PROGRAM PRG_GMD
VAR
END_VAR


// PIP_Gamma Pumps

fb_PCPM3B_PIP_1(i_stGauge := fb_IM2K0_XTES_GCC_1.PG);

// FB_MKS317

fb_EM1K0_GMD_GPI_10(PG=>);
fb_EM1K0_GMD_GPI_40(PG=>);
fb_EM1K0_GMD_GPI_70(PG=>);
fb_IM2K0_XTES_GPI_1(PG=>);
fb_TV1K0_GAS_GPI_1(PG=>);

// FB_PTM_TwisTorr

fb_EM1K0_GMD_PTM_10(i_xExtILKOk := TRUE);
fb_EM1K0_GMD_PTM_20(i_xExtILKOk := TRUE);
fb_EM1K0_GMD_PTM_30(i_xExtILKOk := TRUE);
fb_EM1K0_GMD_PTM_40(i_xExtILKOk := TRUE);
fb_EM1K0_GMD_PTM_50(i_xExtILKOk := TRUE);
fb_EM1K0_GMD_PTM_60(i_xExtILKOk := TRUE);
fb_EM1K0_GMD_PTM_70(i_xExtILKOk := TRUE);

// FB_VRC

fb_EM1K0_GMD_VRC_10(i_xExtILK_OK := TRUE, i_xOverrideMode := xSystemOverrideMode);
fb_EM1K0_GMD_VRC_20(i_xExtILK_OK := TRUE, i_xOverrideMode := xSystemOverrideMode);
fb_EM1K0_GMD_VRC_30(i_xExtILK_OK := TRUE, i_xOverrideMode := xSystemOverrideMode);
fb_EM1K0_GMD_VRC_50(i_xExtILK_OK := TRUE, i_xOverrideMode := xSystemOverrideMode);
fb_EM1K0_GMD_VRC_60(i_xExtILK_OK := TRUE, i_xOverrideMode := xSystemOverrideMode);
fb_EM1K0_GMD_VRC_70(i_xExtILK_OK := TRUE, i_xOverrideMode := xSystemOverrideMode);

// FB_MKS422

fb_EM1K0_GMD_GCC_10(PG := fb_EM1K0_GMD_GPI_10.PG);
fb_EM1K0_GMD_GCC_20(PG := fb_EM1K0_GMD_GPI_10.PG);
fb_EM1K0_GMD_GCC_30(PG := fb_EM1K0_GMD_GPI_10.PG);
fb_EM1K0_GMD_GCC_40(PG := fb_EM1K0_GMD_GPI_40.PG);
fb_EM1K0_GMD_GCC_50(PG := fb_EM1K0_GMD_GPI_70.PG);
fb_EM1K0_GMD_GCC_60(PG := fb_EM1K0_GMD_GPI_70.PG);
fb_EM1K0_GMD_GCC_70(PG := fb_EM1K0_GMD_GPI_70.PG);
fb_IM2K0_XTES_GCC_1(PG := fb_IM2K0_XTES_GPI_1.PG);
fb_TV1K0_GAS_GCC_1(PG := fb_TV1K0_GAS_GPI_1.PG);

// FB_EbaraEVA

fb_EM1K0_GMD_PRT_40(i_xExtIlkOK := TRUE);

END_PROGRAM

(* stored: Version 1.1.0.1, ProductVersion 3.1.4022.12
   POU PRG_GMD: Id {7db60d79-1d43-443c-b047-ee270d12fe07}, SpecialFunc None *)
